FUNCTION_BLOCK L0_State (* Basic Function Block Type *)
  (* Standard: 61499-2; Description: Basic FB to handle CNC service status *)
  (* Version 0.0, 2014-08-25, EQUEROL, UJI *)
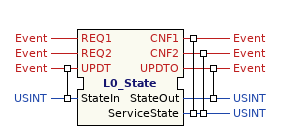
  EVENT_INPUT
    REQ1; (* Request CNC state *)
    REQ2; (* Request CNC state *)
    UPDT WITH StateIn; (* Service state update request *)
  END_EVENT
  EVENT_OUTPUT
    CNF1 WITH ServiceState; (* Execution Confirmation *)
    CNF2 WITH ServiceState; (* Execution Confirmation *)
    UPDTO WITH StateOut; (* CNC state Update indication *)
  END_EVENT
  VAR_INPUT
    StateIn : USINT; (* CNC state enumeration *)
  END_VAR
  VAR_OUTPUT
    StateOut : USINT := 0; (* CNC state enumeration *)
    ServiceState : USINT := 0; (* CNC service state enumeration *)
  END_VAR
  VAR
    CNCState : USINT := 0; (* Current CNC state *)
    CurrentServiceState : USINT := 0; (* Current CNC service state *)
  END_VAR
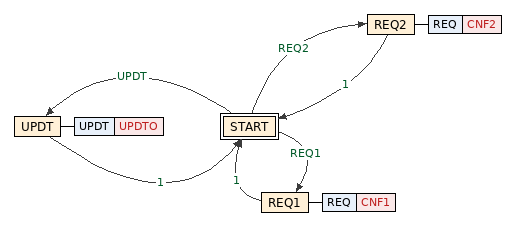
  EC_STATES
    START; (* Initial State *)
    REQ1 : REQ -> CNF1; (* Normal execution *)
    UPDT : UPDT -> UPDTO;
    REQ2 : REQ -> CNF2;
  END_STATES
  EC_TRANSITIONS
    REQ1 TO START := 1;
    START TO REQ1 := REQ1;
    UPDT TO START := 1;
    START TO UPDT := UPDT;
    START TO REQ2 := REQ2;
    REQ2 TO START := 1;
  END_TRANSITIONS
  ALGORITHM REQ IN ST: (* Normally executed algorithm *)
ServiceState := CurrentServiceState;
  END_ALGORITHM
  ALGORITHM UPDT IN ST: (* CNC State update algorithm *)
CNCState := StateIn;
StateOut := CNCState;
IF(CNCState = 1) THEN
	CurrentServiceState := 1;
ELSIF (CNCState = 2) THEN
	CurrentServiceState := 2;
ELSE
	CurrentServiceState := 0;
END_IF;
  END_ALGORITHM
END_FUNCTION_BLOCK
